// TIA Portal project "Complex Object Oriented Programming" (V16)

(* hardware
DEVICE "S71500/ET200MP station_1"  S7-1500 station
   slot 0: "Rail_0"  Rack  6ES7 590-1***0-0AA0
   slot 1: "Control"  CPU 1511-1 PN  6ES7 511-1AK01-0AB0  V2.8
      slot 3: "CPU display_1"  6ES7591-1AA00-0AA0
      slot 32768: "PROFINET interface_1"  X1
         slot 32769: "Port_1"  X1 P1
         slot 32770: "Port_2"  X1 P2
      slot 34817: "Virtual CP interface port_1"  Virtual CP interface port  Virtual CP interface port
DEVICE "SCADA"  SIMATIC PC station
   slot 0: "SIMATIC PC station"  Rail  SIMATIC PC-Station  V1.0
      slot 125: "Stationmanager"  Station_Manager  V6.0.4
   slot 1: "HMI_RT_1"  WinCC RT Professional  6AV2 105-0xxxx-xxxx  16.0.0.0
*)

// ===== PLC "Control"  CPU 1511-1 PN =====

VAR_GLOBAL   // PLC tag table "Auto_Tag"
   "START" AT %M0.0 : Bool;
   "STOP" AT %M0.1 : Bool;
   "LO" AT %M0.2 : Bool;
   "HI" AT %M0.3 : Bool;
   "M_1" AT %M0.4 : Bool;
   "M_2" AT %M0.5 : Bool;
   "M_3" AT %M0.6 : Bool;
   "S0" AT %M0.7 : Bool;
   "S1" AT %M1.0 : Bool;
   "S2" AT %M1.1 : Bool;
   "S3" AT %M1.2 : Bool;
   "T00" AT %M1.3 : Bool;
   "T01" AT %M1.4 : Bool;
   "T12" AT %M1.5 : Bool;
   "T23" AT %M1.6 : Bool;
   "T31" AT %M1.7 : Bool;
   "T10" AT %M2.0 : Bool;
   "T20" AT %M2.1 : Bool;
   "T30" AT %M2.2 : Bool;
   "System_Byte" AT %MB10 : Byte;
   "FirstScan" AT %M10.0 : Bool;
   "DiagStatusUpdate" AT %M10.1 : Bool;
   "AlwaysTRUE" AT %M10.2 : Bool;
   "AlwaysFALSE" AT %M10.3 : Bool;
   "LEVEL" AT %MW20 : Int;
   "Clock_Byte" AT %MB11 : Byte;
   "Clock_10Hz" AT %M11.0 : Bool;
   "Clock_5Hz" AT %M11.1 : Bool;
   "Clock_2.5Hz" AT %M11.2 : Bool;
   "Clock_2Hz" AT %M11.3 : Bool;
   "Clock_1.25Hz" AT %M11.4 : Bool;
   "Clock_1Hz" AT %M11.5 : Bool;
   "Clock_0.625Hz" AT %M11.6 : Bool;
   "Clock_0.5Hz" AT %M11.7 : Bool;
END_VAR

VAR_GLOBAL CONSTANT   // PLC tag table "Auto_Tag"
   "None(1)" : Pip := 65535;
   "Automatic update(1)" : Pip := 0;
   "PIP 1(1)" : Pip := 1;
   "PIP 2(1)" : Pip := 2;
   "PIP 3(1)" : Pip := 3;
   "PIP 4(1)" : Pip := 4;
   "PIP 5(1)" : Pip := 5;
   "PIP 6(1)" : Pip := 6;
   "PIP 7(1)" : Pip := 7;
   "PIP 8(1)" : Pip := 8;
   "PIP 9(1)" : Pip := 9;
   "PIP 10(1)" : Pip := 10;
   "PIP 11(1)" : Pip := 11;
   "PIP 12(1)" : Pip := 12;
   "PIP 13(1)" : Pip := 13;
   "PIP 14(1)" : Pip := 14;
   "PIP 15(1)" : Pip := 15;
   "PIP 16(1)" : Pip := 16;
   "PIP 17(1)" : Pip := 17;
   "PIP 18(1)" : Pip := 18;
   "PIP 19(1)" : Pip := 19;
   "PIP 20(1)" : Pip := 20;
   "PIP 21(1)" : Pip := 21;
   "PIP 22(1)" : Pip := 22;
   "PIP 23(1)" : Pip := 23;
   "PIP 24(1)" : Pip := 24;
   "PIP 25(1)" : Pip := 25;
   "PIP 26(1)" : Pip := 26;
   "PIP 27(1)" : Pip := 27;
   "PIP 28(1)" : Pip := 28;
   "PIP 29(1)" : Pip := 29;
   "PIP 30(1)" : Pip := 30;
   "PIP 31(1)" : Pip := 31;
   "PIP OB Servo(1)" : Pip := 32768;
   "Local~MC(1)" : Hw_SubModule := 51;
   "Local~Common(1)" : Hw_SubModule := 50;
   "Local~Device(1)" : Hw_Device := 32;
   "Local~Configuration(1)" : Hw_SubModule := 33;
   "Local~Display(1)" : Hw_SubModule := 54;
   "Local~Exec(1)" : Hw_SubModule := 52;
   "Local(1)" : Hw_SubModule := 49;
   "Local~PROFINET_interface_1(1)" : Hw_Interface := 64;
   "Local~PROFINET_interface_1~Port_1(1)" : Hw_Interface := 65;
   "Local~PROFINET_interface_1~Port_2(1)" : Hw_Interface := 66;
   "Local~Virtual_communication_interface(1)" : Hw_Interface := 135;
   "OB_Main" : OB_PCYCLE := 1;
   "OB_SIM" : OB_PCYCLE := 123;
END_VAR

DATA_BLOCK "Motor_1"   // DB1
{ S7_Optimized_Access := 'FALSE' }
VERSION : 0.1
// stored: InstanceOfName Motor
"Motor"
BEGIN
END_DATA_BLOCK

DATA_BLOCK "Motor_2"   // DB2
{ S7_Optimized_Access := 'FALSE' }
VERSION : 0.1
// stored: InstanceOfName Motor
"Motor"
BEGIN
END_DATA_BLOCK

DATA_BLOCK "Motor_3"   // DB3
{ S7_Optimized_Access := 'FALSE' }
VERSION : 0.1
// stored: InstanceOfName Motor
"Motor"
BEGIN
END_DATA_BLOCK

// folder: System blocks/Program resources

DATA_BLOCK "T10S"   // DB5
{ S7_Optimized_Access := 'TRUE' }
AUTHOR : Simatic
FAMILY : IEC
NAME : IEC_TMR
VERSION : 1.0
// stored: InstanceOfName IEC_TIMER
"IEC_TIMER"
BEGIN
END_DATA_BLOCK

// folder: (top level)

ORGANIZATION_BLOCK "P&ID"   // OB1, FBD, ProgramCycle
TITLE = "Main Program Sweep (Cycle)"
{ S7_Optimized_Access := 'TRUE' }
VERSION : 0.1
   VAR_INPUT
      Initial_Call : Bool;   // Initial call of this OB
      Remanence : Bool;   // =True, if remanent data are available
   END_VAR
BEGIN

REGION Network 1
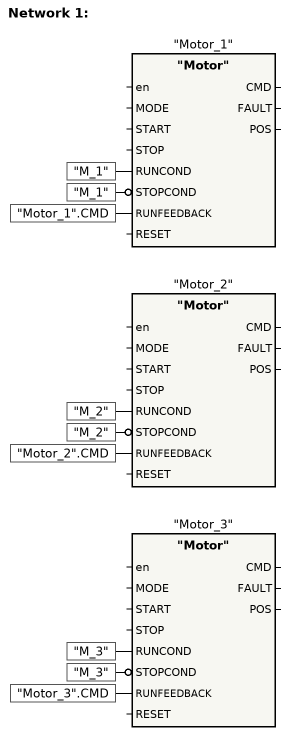
   "Motor_1"(RUNCOND := "M_1", STOPCOND := NOT "M_1", RUNFEEDBACK := "Motor_1".CMD);   // "Motor"
   "Motor_2"(RUNCOND := "M_2", STOPCOND := NOT "M_2", RUNFEEDBACK := "Motor_2".CMD);   // "Motor"
   "Motor_3"(RUNCOND := "M_3", STOPCOND := NOT "M_3", RUNFEEDBACK := "Motor_3".CMD);   // "Motor"
END_REGION
END_ORGANIZATION_BLOCK

ORGANIZATION_BLOCK "SIM"   // OB123, SCL, ProgramCycle
TITLE = "Main Program Sweep (Cycle)"
{ S7_Optimized_Access := 'TRUE' }
VERSION : 0.1
   VAR_INPUT
      Initial_Call : Bool;   // Initial call of this OB
      Remanence : Bool;   // =True, if remanent data are available
   END_VAR
BEGIN
   "R_TRIG_DB"(CLK:="Clock_2Hz");


   IF "Motor_1".RUNFEEDBACK AND "R_TRIG_DB".Q THEN
       "LEVEL" := "LEVEL" + 1;
       IF "LEVEL" >= 100 THEN
           "LEVEL" := 100;
       END_IF;
   END_IF;

   IF "Motor_2".RUNFEEDBACK AND "R_TRIG_DB".Q THEN
       "LEVEL" := "LEVEL" + 1;
       IF "LEVEL" >= 100 THEN
           "LEVEL" := 100;
       END_IF;
   END_IF;

   IF "Motor_3".RUNFEEDBACK AND "R_TRIG_DB".Q THEN
       "LEVEL" := "LEVEL" - 2;
       IF "LEVEL" <= 0 THEN
           "LEVEL" :=0;
       END_IF;
   END_IF;

   IF "LEVEL" >= 99 THEN
       "HI" := TRUE;
   ELSE
       "HI" := FALSE;
   END_IF;

   IF "LEVEL" <= 2 THEN
       "LO" := TRUE;
   ELSE
       "LO" := FALSE;
   END_IF;
END_ORGANIZATION_BLOCK

ORGANIZATION_BLOCK "Auto"   // OB124, SCL, ProgramCycle
TITLE = "Main Program Sweep (Cycle)"
{ S7_Optimized_Access := 'TRUE' }
VERSION : 0.1
   VAR_INPUT
      Initial_Call : Bool;   // Initial call of this OB
      Remanence : Bool;   // =True, if remanent data are available
   END_VAR
BEGIN
   "T10S".TON(IN:="S1",
              PT:=T#10S);

   // TRANSITION EQUATIONS
   // 
   "T00" := "FirstScan";
   "T01" := "S0" AND "START";
   "T12" := "S1" AND "T10S".Q;
   "T23" := "S2" AND "HI";
   "T31" := "S3" AND "LO";
   "T10" := "S1" AND "STOP";
   "T20" := "S2" AND "STOP";
   "T30" := "S3" AND "STOP";

   // STATE EQUATIONS
   // 
   "S0" := ("S0" OR "T00" OR "T10" OR "T20" OR "T30") AND NOT "T01";
   "S1" := ("S1" OR "T01" OR "T31") AND NOT "T12" AND NOT "T10";
   "S2" := ("S2" OR "T12") AND NOT"T23" AND NOT "T20";
   "S3" := ("S3" OR "T23") AND NOT "T31" AND NOT "T30";

   // OUTPUT EQUATIONS
   // 
   "M_1" := "S1" OR "S2";
   "M_2" := "S2";
   "M_3" := "S3";
END_ORGANIZATION_BLOCK

// folder: Lib

FUNCTION_BLOCK "Motor"   // FB1, SCL
{ S7_Optimized_Access := 'FALSE' }
VERSION : 0.1
   VAR_INPUT
      MODE : Int;
      START : Bool;
      STOP : Bool;
      RUNCOND : Bool;
      STOPCOND : Bool;
      RUNFEEDBACK : Bool;
      RESET : Bool;
   END_VAR
   VAR_OUTPUT
      CMD : Bool;
      FAULT : Bool;
      POS : Int;
   END_VAR
   VAR
      Delay : TON_TIME;
      PosCounter : CTU_INT;
      R_TRIG_Instance : R_TRIG;
   END_VAR
BEGIN
   IF #MODE = 1 THEN
       #CMD := (#CMD OR #START) AND NOT #STOP AND NOT #FAULT;
   END_IF;

   IF #MODE = 2 THEN
       #CMD := (#CMD OR #RUNCOND) AND NOT #STOPCOND AND NOT #FAULT;
   END_IF;

   #Delay(IN:=#CMD, PT:= t#5s);

   IF #Delay.Q AND NOT #RUNFEEDBACK THEN
       #FAULT := 1;
   END_IF;

   IF #RESET THEN
       #FAULT := 0;
   END_IF;

   #R_TRIG_Instance(CLK:="Clock_1Hz");

   #PosCounter(CU:=#RUNFEEDBACK AND #R_TRIG_Instance.Q,
               PV:=5,R:= #PosCounter.QU);
   #POS := #PosCounter.CV;
END_FUNCTION_BLOCK

(* ===== HMI "HMI_RT_1" =====
system functions are stored by id; their names below are inferred from use
connection "Connection_1": S71200_TCP_IP, SCADA_S7_1500_OMS

HMI tags "Default tag table"
   "Motor_1" : b3055bf3-543a-47d0-903c-e970704fb603 AT %DB1.DBX0.0, 500 ms
   "Motor_2" : b3055bf3-543a-47d0-903c-e970704fb603 AT %DB2.DBX0.0, 500 ms
   "Motor_3" : b3055bf3-543a-47d0-903c-e970704fb603 AT %DB3.DBX0.0, 500 ms
   "Start" : Bool AT %M0.0, 500 ms
   "Stop" : Bool AT %M0.1, 500 ms
   "Level" : Int AT %MW20, 500 ms

screen "Motor" 300x200
   Button "Button_1" at 26,88 size 80x30; TextOff 'Start'
      on PressLeft: SetBit(".Start")
      on ReleaseLeft: ResetBit(".Start")
   ComboBox "Combo box_1" at 32,28 size 161x38; Text0 'Manual'; Text1 'Auto'
      SelectedIndex <- ".Mode"
   Button "Button_2" at 123,90 size 80x30; TextOff 'Stop'
      on PressLeft: SetBit(".Stop")
      on ReleaseLeft: ResetBit(".Stop")
   Circle "Circle_1" at 90,131 size 59x59
      Appearance <- ".RunFeedback"
   Circle "Circle_2" at 134,161 size 23x23
      Appearance <- ".Fault"
      Visibility <- ".Fault"
   Button "Button_3" at 171,140 size 80x30; TextOff 'Reset'
      on PressLeft: SetBit(".Reset")
      on ReleaseLeft: ResetBit(".Reset")
   GraphicView "Graphic view_1" at 270,6 size 26x22; Picture "Graphic_1"
      on Click: ResetBit(".Show")

screen "Main" 1024x768
   ScreenWindow "Screen window_1" at 41,23 size 320x220; ScreenName "Motor"
      Visibility <- "Show"
   ScreenWindow "Screen window_2" at 63,399 size 320x220; ScreenName "Motor"
      Visibility <- "Show"
   ScreenWindow "Screen window_3" at 676,93 size 320x220; ScreenName "Motor"
      Visibility <- "Show"
   TubePolyline "Pipe_1" at 296,265 size 180x4
   TubePolyline "Pipe_2" at 296,637 size 180x4
   TubePolyline "Pipe_3" at 584,429 size 180x4
   SymbolLibrary "Symbol library_1" at 212,225 size 120x120
      Appearance <- "RunFeedback"
      on Click: InvertBit("Show")
   SymbolLibrary "Symbol library_2" at 212,591 size 120x120
      on Click: InvertBit("Show")
      Appearance <- "RunFeedback"
   SymbolLibrary "Symbol library_3" at 733,370 size 120x120
      on Click: InvertBit("Show")
      Appearance <- "RunFeedback"
   SymbolLibrary "Symbol library_4" at 405,131 size 265x609
   Bar "Bar_1" at 464,193 size 100x517; MinimumValue 0; MaximumValue 100
      ProcessValue <- "Level"
   Button "Button_2" at 811,602 size 80x30; TextOff 'Stop'
      on PressLeft: SetBit("Stop")
      on ReleaseLeft: ResetBit("Stop")
   Button "Button_1" at 717,602 size 80x30; TextOff 'Start'
      on PressLeft: SetBit("Start")
      on ReleaseLeft: ResetBit("Start")
*)